TYPE E_SeasonPL : (Wiosna:=1, Lato, Jesien, Zima);
END_TYPE

(* stored: Version 1.1.0.1, ProductVersion 3.1.4019.2
   DUT E_SeasonPL: Id {e989e0f3-56a8-4563-90de-9cd8719dfd5c} *)
